// TIA Portal V18 export
// export: Created 2026-06-11T19:04:15.6170586Z, ExportSetting WithDefaults, DisplayName Totally Integrated Automation Portal, DisplayVersion V18, DisplayName TIA Portal Openness, DisplayVersion V18, DisplayName TIA Portal Version Control Interface, DisplayVersion V18, DisplayName STEP 7 Professional, DisplayVersion V18, DisplayName STEP 7 Safety, DisplayVersion V18, DisplayName WinCC Professional, DisplayVersion V18
Screen "scadabai7"  1920x1080, Number=8
  ScreenLayer 
    GraphicView "Graphic view_1" at 0,0 size 1290x766  Picture=nen_3
    IOField "I/O field_1" at 30,69 size 59x14  DataFormat=Decimal, FormatPattern=9999999999, Mode=InOutput
    IOField "I/O field_2" at 226,69 size 51x15  DataFormat=Decimal, FormatPattern=9999999999, Mode=InOutput
    IOField "I/O field_3" at 226,213 size 53x15  DataFormat=Decimal, FormatPattern=9999999999, Mode=InOutput
    IOField "I/O field_4" at 31,207 size 58x15  DataFormat=Decimal, FormatPattern=9999999999, Mode=InOutput
    IOField "I/O field_5" at 225,103 size 51x15  DataFormat=Decimal, FormatPattern=9999999999, Mode=InOutput
    IOField "I/O field_6" at 418,105 size 54x14  DataFormat=Decimal, FormatPattern=9999999999, Mode=InOutput
    IOField "I/O field_7" at 421,286 size 53x15  DataFormat=Decimal, FormatPattern=9999999999, Mode=InOutput
    IOField "I/O field_8" at 421,317 size 55x15  DataFormat=Decimal, FormatPattern=9999999999, Mode=InOutput
    IOField "I/O field_9" at 641,232 size 55x15  DataFormat=Decimal, FormatPattern=9999999999, Mode=InOutput
    IOField "I/O field_10" at 641,258 size 56x15  DataFormat=Decimal, FormatPattern=9999999999, Mode=InOutput
    IOField "I/O field_11" at 603,292 size 53x15  DataFormat=Decimal, FormatPattern=9999999999, Mode=InOutput
    IOField "I/O field_12" at 442,387 size 27x11  DataFormat=Decimal, FormatPattern=9999999999, Mode=InOutput
    IOField "I/O field_13" at 442,399 size 26x11  DataFormat=Decimal, FormatPattern=9999999999, Mode=InOutput
    IOField "I/O field_14" at 442,411 size 27x11  DataFormat=Decimal, FormatPattern=9999999999, Mode=InOutput
    IOField "I/O field_15" at 421,442 size 47x11  DataFormat=Decimal, FormatPattern=9999999999, Mode=InOutput
    IOField "I/O field_16" at 623,366 size 29x11  DataFormat=Decimal, FormatPattern=9999999999, Mode=InOutput
    IOField "I/O field_17" at 623,379 size 28x11  DataFormat=Decimal, FormatPattern=9999999999, Mode=InOutput
    IOField "I/O field_18" at 623,390 size 29x11  DataFormat=Decimal, FormatPattern=9999999999, Mode=InOutput
    IOField "I/O field_19" at 554,501 size 28x11  DataFormat=Decimal, FormatPattern=9999999999, Mode=InOutput
    IOField "I/O field_20" at 261,531 size 56x11  DataFormat=Decimal, FormatPattern=9999999999, Mode=InOutput
    IOField "I/O field_21" at 99,531 size 58x11  DataFormat=Decimal, FormatPattern=9999999999, Mode=InOutput
    IOField "I/O field_22" at 14,477 size 51x11  DataFormat=Decimal, FormatPattern=9999999999, Mode=InOutput
    IOField "I/O field_23" at 554,512 size 28x11  DataFormat=Decimal, FormatPattern=9999999999, Mode=InOutput
    IOField "I/O field_24" at 554,523 size 28x11  DataFormat=Decimal, FormatPattern=9999999999, Mode=InOutput
    IOField "I/O field_25" at 1014,533 size 34x11  DataFormat=Decimal, FormatPattern=9999999999, Mode=InOutput
    IOField "I/O field_26" at 1014,545 size 34x11  DataFormat=Decimal, FormatPattern=9999999999, Mode=InOutput
    IOField "I/O field_27" at 1014,557 size 34x11  DataFormat=Decimal, FormatPattern=9999999999, Mode=InOutput
    IOField "I/O field_28" at 1100,556 size 53x11  DataFormat=Decimal, FormatPattern=9999999999, Mode=InOutput
    IOField "I/O field_29" at 857,345 size 57x11  DataFormat=Decimal, FormatPattern=9999999999, Mode=InOutput
    IOField "I/O field_30" at 857,274 size 56x11  DataFormat=Decimal, FormatPattern=9999999999, Mode=InOutput
    TextField "Text field_1" at 92,69 size 34x11  Text="Kgf/cm2"
    GraphicView "Graphic view_2" at 147,130 size 66x47  Picture=bon 1
    GraphicView "Graphic view_3" at 97,88 size 22x16  Picture=Graphic_32
    GraphicView "Graphic view_4" at 97,119 size 22x16  Picture=Graphic_32
    GraphicView "Graphic view_5" at 97,175 size 22x16  Picture=Graphic_32
    GraphicView "Graphic view_6" at 546,176 size 22x16  Picture=Graphic_32
    GraphicView "Graphic view_7" at 546,119 size 22x16  Picture=Graphic_32
    GraphicView "Graphic view_8" at 639,340 size 25x16  Picture=Graphic_32
    Rectangle "Rectangle_1" at 28,416 size 14x13
    Rectangle "Rectangle_2" at 122,416 size 14x13
    Rectangle "Rectangle_3" at 216,416 size 14x13
    Rectangle "Rectangle_4" at 310,416 size 14x13
    Rectangle "Rectangle_5" at 961,369 size 14x13
    Rectangle "Rectangle_6" at 774,636 size 13x11
    IOField "I/O field_31" at 857,230 size 56x11  DataFormat=Decimal, FormatPattern=9999999999, Mode=InOutput
    IOField "I/O field_32" at 856,155 size 58x11  DataFormat=Decimal, FormatPattern=9999999999, Mode=InOutput
    IOField "I/O field_33" at 856,116 size 57x11  DataFormat=Decimal, FormatPattern=9999999999, Mode=InOutput
    IOField "I/O field_34" at 1033,54 size 85x15  DataFormat=Decimal, FormatPattern=9999999999, Mode=InOutput
    IOField "I/O field_35" at 1033,74 size 85x15  DataFormat=Decimal, FormatPattern=9999999999, Mode=InOutput
    IOField "I/O field_36" at 1033,94 size 85x15  DataFormat=Decimal, FormatPattern=9999999999, Mode=InOutput
    Circle "Circle_1" at 1035,361 size 15x15
    Ellipse "Ellipse_1" at 1032,378 size 22x18
    GraphicView "Graphic view_9" at 957,380 size 24x16  Picture=Graphic_32
    GraphicView "Graphic view_10" at 1032,508 size 24x16  Picture=Graphic_32
    GraphicView "Graphic view_11" at 1156,508 size 24x16  Picture=Graphic_32
    GraphicView "Graphic view_12" at 1104,576 size 24x16  Picture=Graphic_32
    GraphicView "Graphic view_13" at 747,626 size 24x16  Picture=Graphic_32
    GraphicView "Graphic view_14" at 747,585 size 24x16  Picture=Graphic_32
    Ellipse "Ellipse_2" at 439,569 size 19x16
    Ellipse "Ellipse_3" at 439,619 size 19x16
    Ellipse "Ellipse_4" at 519,600 size 15x13
    Ellipse "Ellipse_5" at 273,417 size 15x13
    Ellipse "Ellipse_6" at 366,416 size 15x13
    IOField "I/O field_37" at 210,477 size 49x11  DataFormat=Decimal, FormatPattern=9999999999, Mode=InOutput
    Button "Button_1" at 1040,119 size 69x28  Mode=Text, TextOff="Tank status", TextOn="Text"
    Button "Button_2" at 1138,142 size 54x21  Mode=Text, TextOff="Start", TextOn="Text"
    Button "Button_3" at 1220,60 size 54x22  Mode=Text, TextOff="Manual", TextOn="Text"
    Button "Button_4" at 1139,60 size 54x23  Mode=Text, TextOff="Auto", TextOn="Text"
    Button "Button_5" at 1220,142 size 54x21  Mode=Text, TextOff="Stop", TextOn="Text"
    Button "Button_6" at 1139,214 size 54x21  Mode=Text, TextOff="Start", TextOn="Text"
    Button "Button_7" at 1219,214 size 54x21  Mode=Text, TextOff="Stop", TextOn="Text"
    Button "Button_8" at 1139,454 size 54x21  Mode=Text, TextOff="Start", TextOn="Text"
    Button "Button_9" at 1219,454 size 54x21  Mode=Text, TextOff="Stop", TextOn="Text"
    Button "Button_10" at 1136,479 size 70x21  Mode=Text, TextOff="Process Over", TextOn="Text"
    IOField "I/O field_38" at 1218,106 size 38x15  DataFormat=Decimal, FormatPattern=9999999999, Mode=InOutput
    IOField "I/O field_39" at 1218,125 size 38x12  DataFormat=Decimal, FormatPattern=9999999999, Mode=InOutput
    IOField "I/O field_40" at 1218,177 size 38x12  DataFormat=Decimal, FormatPattern=9999999999, Mode=InOutput
    IOField "I/O field_41" at 1217,197 size 38x12  DataFormat=Decimal, FormatPattern=9999999999, Mode=InOutput
    IOField "I/O field_42" at 1218,257 size 38x12  DataFormat=Decimal, FormatPattern=9999999999, Mode=InOutput
    IOField "I/O field_43" at 1218,301 size 38x12  DataFormat=Decimal, FormatPattern=9999999999, Mode=InOutput
    IOField "I/O field_44" at 1218,320 size 38x12  DataFormat=Decimal, FormatPattern=9999999999, Mode=InOutput
    IOField "I/O field_45" at 1218,339 size 38x12  DataFormat=Decimal, FormatPattern=9999999999, Mode=InOutput
    IOField "I/O field_46" at 1218,358 size 38x12  DataFormat=Decimal, FormatPattern=9999999999, Mode=InOutput
    IOField "I/O field_47" at 1189,437 size 31x12  DataFormat=Decimal, FormatPattern=9999999999, Mode=InOutput
    IOField "I/O field_48" at 1247,438 size 17x12  DataFormat=Decimal, FormatPattern=9999999999, Mode=InOutput
    IOField "I/O field_49" at 994,331 size 49x14  DataFormat=Decimal, FormatPattern=9999999999, Mode=InOutput
    IOField "I/O field_50" at 994,345 size 49x12  DataFormat=Decimal, FormatPattern=9999999999, Mode=InOutput
    IOField "I/O field_51" at 845,624 size 62x11  DataFormat=Decimal, FormatPattern=9999999999, Mode=InOutput
    IOField "I/O field_52" at 845,654 size 62x11  DataFormat=Decimal, FormatPattern=9999999999, Mode=InOutput
    IOField "I/O field_53" at 846,685 size 62x11  DataFormat=Decimal, FormatPattern=9999999999, Mode=InOutput
    IOField "I/O field_54" at 957,624 size 62x11  DataFormat=Decimal, FormatPattern=9999999999, Mode=InOutput
    IOField "I/O field_55" at 956,654 size 62x11  DataFormat=Decimal, FormatPattern=9999999999, Mode=InOutput
    IOField "I/O field_56" at 956,685 size 55x11  DataFormat=Decimal, FormatPattern=9999999999, Mode=InOutput
    IOField "I/O field_57" at 1068,685 size 93x11  DataFormat=Decimal, FormatPattern=9999999999, Mode=InOutput
    IOField "I/O field_58" at 1069,624 size 91x11  DataFormat=Decimal, FormatPattern=9999999999, Mode=InOutput
    IOField "I/O field_59" at 1069,654 size 60x11  DataFormat=Decimal, FormatPattern=9999999999, Mode=InOutput
    IOField "I/O field_60" at 1198,614 size 71x11  DataFormat=Decimal, FormatPattern=9999999999, Mode=InOutput
    IOField "I/O field_62" at 1184,654 size 54x11  DataFormat=Decimal, FormatPattern=9999999999, Mode=InOutput
    IOField "I/O field_63" at 1182,684 size 90x11  DataFormat=Decimal, FormatPattern=9999999999, Mode=InOutput
    IOField "I/O field_61" at 1198,626 size 31x11  DataFormat=Decimal, FormatPattern=9999999999, Mode=InOutput
    TextField "Text field_2" at 92,208 size 30x11  Text="Deg C."
    TextField "Text field_3" at 287,69 size 30x11  Text="Deg C."
    TextField "Text field_4" at 286,104 size 30x11  Text="Deg C."
    TextField "Text field_5" at 286,213 size 30x11  Text="Deg C."
    TextField "Text field_6" at 478,104 size 34x11  Text="Kgf/cm2"
    TextField "Text field_7" at 488,287 size 12x11  Text="Vh"
    TextField "Text field_8" at 488,318 size 27x11  Text="Kg/m3"
    TextField "Text field_10" at 73,477 size 12x11  Text="cm"
    TextField "Text field_11" at 168,530 size 12x11  Text="cm"
    TextField "Text field_12" at 274,475 size 12x11  Text="cm"
    TextField "Text field_13" at 331,528 size 12x11  Text="cm"
    TextField "Text field_14" at 702,232 size 12x11  Text="Vh"
    TextField "Text field_15" at 704,260 size 27x11  Text="Kg/m3"
    TextField "Text field_16" at 664,293 size 19x11  Text="Kg/h"
    TextField "Text field_17" at 916,116 size 30x11  Text="Deg C."
    TextField "Text field_18" at 916,155 size 30x11  Text="Deg C."
    TextField "Text field_19" at 916,229 size 30x11  Text="Deg C."
    TextField "Text field_20" at 916,274 size 30x11  Text="Deg C."
    TextField "Text field_21" at 918,345 size 30x11  Text="Deg C."
    TextField "Text field_9" at 1049,532 size 19x11  Text="Kg/h"
    TextField "Text field_22" at 1049,543 size 19x11  Text="Kg/h"
    TextField "Text field_23" at 1049,555 size 10x11  Text="%"
    TextField "Text field_24" at 1161,555 size 19x11  Text="Kg/h"
    TextField "Text field_25" at 908,624 size 30x11  Text="Deg C."
    TextField "Text field_26" at 907,653 size 30x11  Text="Deg C."
    TextField "Text field_27" at 907,683 size 30x11  Text="Deg C."
    TextField "Text field_28" at 1018,654 size 30x11  Text="Deg C."
    TextField "Text field_29" at 1024,623 size 19x11  Text="Kg/h"
    TextField "Text field_30" at 1014,684 size 34x11  Text="Kgf/cm2"
    TextField "Text field_31" at 1108,624 size 34x11  Text="Kgf/cm2"
    TextField "Text field_32" at 1130,654 size 30x11  Text="Deg C."
    TextField "Text field_33" at 1125,684 size 34x11  Text="Kgf/cm2"
    TextField "Text field_34" at 1227,613 size 34x11  Text="Kgf/cm2"
    TextField "Text field_35" at 1236,625 size 10x11  Text="%"
    TextField "Text field_36" at 1241,654 size 30x11  Text="Deg C."
    TextField "Text field_37" at 1227,683 size 34x11  Text="Kgf/cm2"
    Button "Button_11" at 18,711 size 37x38  Mode=Text, TextOn="Text"
    Button "Button_12" at 168,711 size 37x38  Mode=Text, TextOn="Text"
    Button "Button_13" at 319,711 size 37x38  Mode=Text, TextOn="Text"
    Button "Button_14" at 473,711 size 37x38  Mode=Text, TextOn="Text"
    Button "Button_15" at 624,712 size 37x38  Mode=Text, TextOn="Text"
    Button "Button_16" at 778,712 size 37x38  Mode=Text, TextOn="Text"
    Button "Button_17" at 928,712 size 37x38  Mode=Text, TextOn="Text"
    GraphicView "Graphic view_15" at 462,575 size 32x26  Picture=Graphic_34
    GraphicView "Graphic view_16" at 462,624 size 32x26  Picture=Graphic_34
    Button "Button_18" at 101,5 size 29x30  Mode=Text, TextOn="Text"
    Button "Button_19" at 154,5 size 29x30  Mode=Text, TextOn="Text"
    Button "Button_20" at 208,5 size 30x30  Mode=Text, TextOn="Text"
    Button "Button_21" at 262,5 size 30x30  Mode=Text, TextOn="Text"
    Button "Button_22" at 315,6 size 30x30  Mode=Text, TextOn="Text"
    IOField "I/O field_64" at 997,7 size 85x15  DataFormat=Decimal, FormatPattern=9999999999, Mode=InOutput
    IOField "I/O field_65" at 997,21 size 85x15  DataFormat=Decimal, FormatPattern=9999999999, Mode=InOutput
    GraphicView "Graphic view_17" at 456,361 size 25x16  Picture=Graphic_32
    GraphicView "Graphic view_18" at 1020,428 size 38x31  Picture=Graphic_35
    Button "Button_23" at 32,296 size 51x17  Mode=Text, TextOff="Open", TextOn="Text"
    Button "Button_24" at 94,296 size 47x17  Mode=Text, TextOff="Close", TextOn="Text"
    Circle "Circle_2" at 137,108 size 10x10
    Circle "Circle_3" at 166,187 size 10x10
    Circle "Circle_4" at 180,85 size 10x10
    Circle "Circle_5" at 343,100 size 10x10
    Circle "Circle_6" at 338,206 size 10x10
    Circle "Circle_7" at 529,100 size 10x10
    Circle "Circle_8" at 597,222 size 10x10
    Circle "Circle_9" at 585,327 size 10x10
    Circle "Circle_10" at 489,341 size 10x10
    Circle "Circle_11" at 405,463 size 10x10
    Circle "Circle_12" at 329,554 size 10x10
    Circle "Circle_13" at 240,555 size 10x10
    Circle "Circle_14" at 150,556 size 10x10
    Circle "Circle_15" at 59,556 size 10x10
    Circle "Circle_16" at 831,114 size 10x10
    Circle "Circle_17" at 831,153 size 10x10
    Circle "Circle_18" at 831,229 size 10x10
    Circle "Circle_19" at 831,271 size 10x10
    Circle "Circle_20" at 899,410 size 10x10
    Circle "Circle_21" at 1092,480 size 10x10
    Button "Btn_Enter_System_4" at 1290,0 size 114x38  Mode=Text, StyleItem=Button, TextOff="Mh login", TextOn="Text"
      VisibilityAnimation "VisibilityAnimation"  RangeEnd=99, RangeStart=1
        tag Logged_In
      on Click: ActivateScreen(Screen name := Login/out, Object number := 0)
    Button "Button_25" at 1079,712 size 37x38  Mode=Text, TextOn="Text"
    Button "Button_26" at 1236,712 size 37x38  Mode=Text, TextOn="Text"
